Omron CX-Programmer project NewProject (CX-Programmer 9.73)

# PLC Tugas_Akhir: CP2E S

## Global symbols (name address type ; comment)
0.00 BOOL  ; PB_Start
0.01 BOOL  ; PB_Stop
0.02 BOOL  ; SENSOR_A
0.03 BOOL  ; SENSOR_B
0.04 BOOL  ; MANIPULATOR_DONE
100.00 BOOL  ; System_Run
100.01 BOOL  ; STEP_A_WAIT
100.02 BOOL  ; STEP_B_WAIT
100.03 BOOL  ; STEP_MANIPULATOR
100.04 BOOL  ; DONE
10.00 BOOL  ; CONVEYOR
10.01 BOOL  ; MANIPULATOR
10.02 BOOL  ; LAMPU_SELESAI

## Program NewProgram1 (cyclic task 0)

### Section Section1

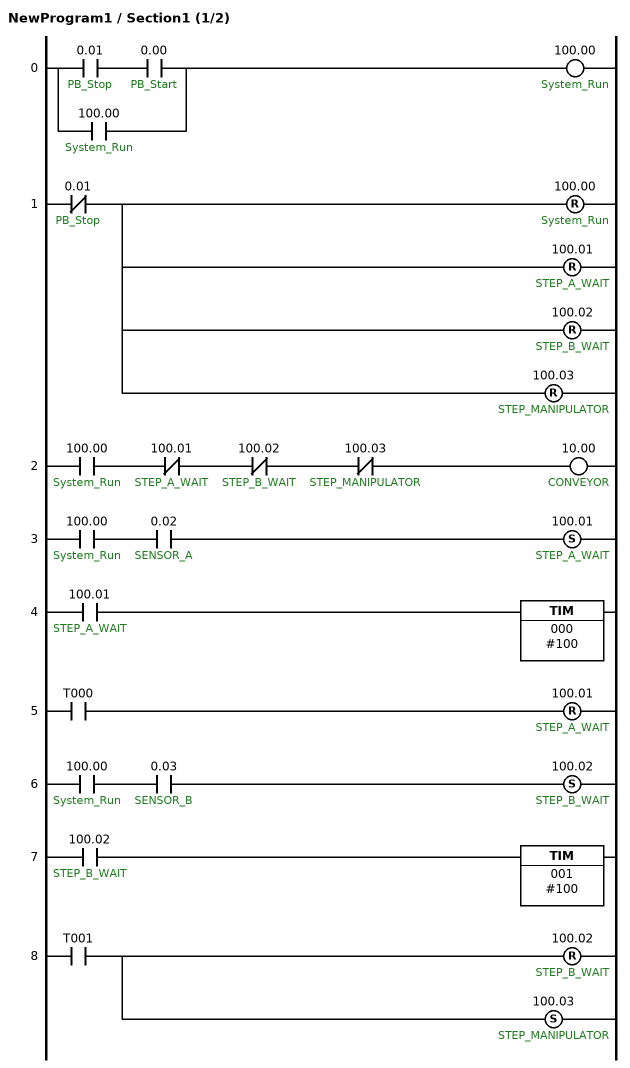
; rung 0
LD 0.01  ; PB_Stop
AND 0.00  ; PB_Start
OR 100.00  ; System_Run
OUT 100.00  ; System_Run
; rung 1
LDNOT 0.01  ; PB_Stop
RSET 100.00  ; System_Run
RSET 100.01  ; STEP_A_WAIT
RSET 100.02  ; STEP_B_WAIT
RSET 100.03  ; STEP_MANIPULATOR
; rung 2
LD 100.00  ; System_Run
ANDNOT 100.01  ; STEP_A_WAIT
ANDNOT 100.02  ; STEP_B_WAIT
ANDNOT 100.03  ; STEP_MANIPULATOR
OUT 10.00  ; CONVEYOR
; rung 3
LD 100.00  ; System_Run
AND 0.02  ; SENSOR_A
SET 100.01  ; STEP_A_WAIT
; rung 4
LD 100.01  ; STEP_A_WAIT
TIM 000 #100
; rung 5
LD T000
RSET 100.01  ; STEP_A_WAIT
; rung 6
LD 100.00  ; System_Run
AND 0.03  ; SENSOR_B
SET 100.02  ; STEP_B_WAIT
; rung 7
LD 100.02  ; STEP_B_WAIT
TIM 001 #100
; rung 8
LD T001
RSET 100.02  ; STEP_B_WAIT
SET 100.03  ; STEP_MANIPULATOR

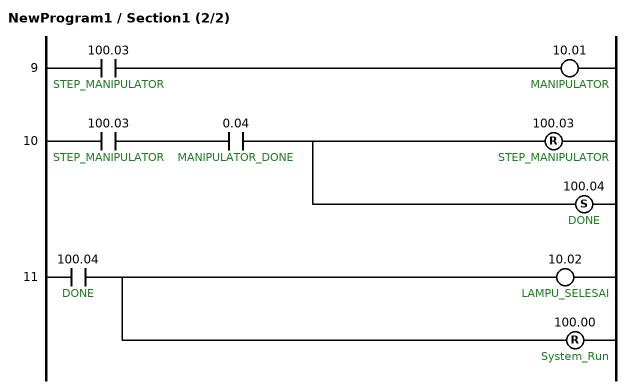
; rung 9
LD 100.03  ; STEP_MANIPULATOR
OUT 10.01  ; MANIPULATOR
; rung 10
LD 100.03  ; STEP_MANIPULATOR
AND 0.04  ; MANIPULATOR_DONE
RSET 100.03  ; STEP_MANIPULATOR
SET 100.04  ; DONE
; rung 11
LD 100.04  ; DONE
OUT 10.02  ; LAMPU_SELESAI
RSET 100.00  ; System_Run

### Section END
; rung 0
END(001)